(* CODESYS project cl_errorsdatabaseplc.library
   Company: CleanGreensSA
   Description: class to load error and class messages from SQL database
   Version: 1.0
   Placeholder: CL_errorDB
   Author: Martin Coffy and Massimo Lucano
   Title: ErrorDatabase_class

Project tree, tasks and I/O mapping:
  libraries: Tc2_Database, * (Beckhoff Automation GmbH); Tc2_DataExchange, * (Beckhoff Automation GmbH); Tc2_Standard, * (Beckhoff Automation GmbH); Tc2_System, * (Beckhoff Automation GmbH); Tc2_Utilities, * (Beckhoff Automation GmbH); Tc3_Database, * (Beckhoff Automation GmbH); Tc3_EventLogger, * (Beckhoff Automation GmbH); Tc3_Module, * (Beckhoff Automation GmbH)
  DUTs/
    Database/
      data type Main_STM
      data type ST_classAndErrorNum
      data type ST_ErrorDBConst
      data type ST_ParameterValues
      data type ST_SP_ClassReturn
      data type ST_SP_RecordReturn
      data type ST_valToAccess
      data type STM_LoadDB
  GVLs/
    global variables C
  POUs/
    Classes_database_connection/
      function block CL_CGSDictionnary [ST]: Init, Search
      function block CL_ErrorDB [ST]: GetClassMsg, GetErrorLongMsg, GetErrorRemedMsg, GetErrorShortMsg, GetNumerics, Init, nextPower2, numIterations, Run, SearchClassData, SearchErrorData, sMsgLang, stConstValues, WhichSeverity
      function block FB_SP_getClassNameAndIDs [ST]
      function block FB_SP_getErrorsMessages [ST]
*)

// DUTs/Database/Main_STM
{attribute 'qualified_only'}
{attribute 'strict'}
TYPE Main_STM :
(
  Init,
  Run,
  FillingArrays,
  SearchIndex,
  Idle,
  Error
);
END_TYPE

// DUTs/Database/ST_classAndErrorNum
TYPE ST_classAndErrorNum :
	STRUCT
		errorId					: STRING(3);
		classId					: STRING(3);
		telegramSending	: STRING(1);
		hmiErrorShow		: STRING(1);
		instanceNum			: BYTE;
	END_STRUCT
END_TYPE

// DUTs/Database/ST_ErrorDBConst
TYPE ST_ErrorDBConst :
	STRUCT
		udiErrNumRecord		  :	UDINT := 0;
		udiClassNumRecord		:	UDINT := 0;
		sLanguageForErrors	:	STRING(2)	:= 'en';
		udiUsedDB						:	UDINT := 0;
		tDBConnectTimeout		:	TIME	:=	TIME#15S;
		tAMSTimeout					:	TIME	:=	TIME#10S;
	END_STRUCT
END_TYPE

// DUTs/Database/ST_ParameterValues
TYPE ST_ParameterValues :
STRUCT
	lang: STRING(2);
END_STRUCT
END_TYPE

// DUTs/Database/ST_SP_ClassReturn
TYPE ST_SP_ClassReturn :
STRUCT
	tableId: UDINT;
	classId: STRING(3);
	className: STRING(255);
	instanceNum: BYTE;
	objDescriptMsg:	STRING(255);
END_STRUCT
END_TYPE

// DUTs/Database/ST_SP_RecordReturn
TYPE ST_SP_RecordReturn :
STRUCT
	tableId: UDINT;
	//classId: STRING(3);
	errorId: STRING(3);
	severity: BYTE;
	errorMsgShort: STRING(255);
	errorMsgLong: STRING(255);
	remediationMsg: STRING(255);
	telegramSending: STRING(1);
	hmiErrorShow: STRING(1);
END_STRUCT
END_TYPE

// DUTs/Database/ST_valToAccess
TYPE ST_valToAccess :
STRUCT
  	severity: BYTE;
	errorSummary:	STRING(255);
	errorMessage: STRING(255);
	remediationMessage: STRING(255);
	telegramSending: STRING(1);
	hmiErrorShow: STRING(1);
END_STRUCT
END_TYPE

// DUTs/Database/STM_LoadDB
{attribute 'qualified_only'}
{attribute 'strict'}
TYPE STM_LoadDB :
(
  
  GetAMSAdress,
	StoreErrorView,
	StoreClassView,
  GenErrorKeys,
	GenClassKeys,
	EndReadingDB
);
END_TYPE

// GVLs/C
// constant to be set in order to describe the greenhouse
// abbreviation GH stands everywhere for Greenhouse
{attribute 'qualified_only'}
VAR_GLOBAL CONSTANT 
  //Errors database constants
  nMaxRecordsDb_C          : UDINT := 1024;
  nMaxUpSize_C             : UDINT := 2048;
  //uiErrorUpSizePowerTwo_C : UDINT := 1024;
  //uiClassUpSizePowerTwo_C : UDINT := 1024;
END_VAR

// POUs/Classes_database_connection/CL_CGSDictionnary
FUNCTION_BLOCK CL_CGSDictionnary
VAR
	bInit	            :	BOOL	:= FALSE;
	
	_usiNbIter_C	    :	USINT;
	_udiSizeKeyArray	:	UDINT;
	
	usiSearchIter     : USINT;
  udiUpId           : UDINT;
  udiDownId         : UDINT;
	
	// Pointer to the keys array to search into
	_udiKeyArray_P	:	POINTER TO UDINT;	// Access to the keys array with a pointer, limited risks as long as udiUpId and udiDownId are correctly set.
END_VAR

METHOD PUBLIC Init : BOOL
VAR_INPUT
	udiKeyArray_P		:	POINTER TO UDINT;
	usiNbIter_C			:	SINT;
	udiSizeKeyArray	:	UDINT;
END_VAR

VAR
	bInputContract 	: BOOL;
END_VAR
Init := FALSE;

IF NOT bInit THEN
		
	bInputContract := 		udiKeyArray_P <> 0
										AND usiNbIter_C > 0 
										AND LREAL_TO_UDINT(EXPT(2,usiNbIter_C)) = udiSizeKeyArray;	// For the real size of the array, to do it outside (too complicated here)
	
	IF bInputContract THEN	// Test for the size of the inputs: to check if possible 
		
		// Initialisation of the "constant" values
		_udiKeyArray_P		:= udiKeyArray_P;
		_usiNbIter_C			:=	usiNbIter_C;
		_udiSizeKeyArray	:= udiSizeKeyArray;
		
		// Initialisation for the method
		usiSearchIter := usiNbIter_C;
  	udiUpId       := udiSizeKeyArray;
  	udiDownId     := 1;
		bInit := TRUE;
	END_IF
END_IF
END_METHOD

METHOD Search : BOOL
VAR_INPUT
  udiKey_DB	:	UDINT	:=	0;
END_VAR
VAR_OUTPUT
	udiFoundKeyIndex	:	UDINT;
  bError:  BOOL;
END_VAR
VAR
  udiMidDownId: UDINT;
  udiMidUpId: UDINT;
  udiMidUpKey: UDINT;
  udiMidLowKey:  UDINT;
END_VAR
IF bInit THEN

  Search := FALSE; 
  bError := FALSE;
  
  udiMidDownId := (udiUpId+udiDownId-1)/2;
  udiMidUpId := udiMidDownId+1;
      
  udiMidUpKey := _udiKeyArray_P[udiMidUpId];
  udiMidLowKey := _udiKeyArray_P[udiMidDownId];
      
  // Also manage the case when final iter and no case found
  IF udiKey_DB = udiMidLowKey THEN
		udiFoundKeyIndex := udiMidDownId+1;	// +1 required, since the Pointer index begins at 0, while the corresponding array starts at 1!
		usiSearchIter := _usiNbIter_C;
		udiUpId   := _udiSizeKeyArray;
		udiDownId := 1;
    Search := TRUE;
  ELSIF udiMidUpKey = udiKey_DB THEN
		udiFoundKeyIndex := udiMidUpId+1;	//+1 required, since the Pointer index begins at 0, while the corresponding array starts at 1!
		usiSearchIter := _usiNbIter_C;
		udiUpId   := _udiSizeKeyArray;
		udiDownId := 1;
    Search	:= TRUE;
  ELSE 
    IF usiSearchIter > 1 THEN
      IF udiMidLowKey > udiKey_DB THEN
          udiUpId := udiMidDownId;
					usiSearchIter := usiSearchIter-1;
      ELSIF udiMidUpKey < udiKey_DB THEN
          udiDownId := udiMidUpId;
					usiSearchIter := usiSearchIter-1;
      ELSE
				usiSearchIter := _usiNbIter_C;
				udiUpId   := _udiSizeKeyArray;
				udiDownId := 1;
				Search := TRUE;
				bError := TRUE;
      END_IF
    ELSE
			usiSearchIter := _usiNbIter_C;
			udiUpId   := _udiSizeKeyArray;
			udiDownId := 1;
      Search := TRUE;
      bError := TRUE;
    END_IF
  END_IF
END_IF
END_METHOD

END_FUNCTION_BLOCK

// POUs/Classes_database_connection/CL_ErrorDB
FUNCTION_BLOCK CL_ErrorDB
VAR  
  // Internal variables
  bInit                   :	BOOL	:= FALSE;
  stmMain                 : Main_STM := Main_STM.Init;
	
	// AMS variable
	fbAMSaddrGetter	        :	FB_GetLocalAmsNetId;
  
  // DB related variables
  // langStruct: ST_ParameterValues := (lang := C.sLangErrors);
  dbErrorConnector        : FB_SP_getErrorsMessages;
	dbClassConnector        :	FB_SP_getClassNameAndIDs;
  stmLoadDB               : STM_LoadDB	:= STM_LoadDB.GetAMSAdress;
  udiIndex                : UDINT := 1;
  
  // Size-related variables (previously known)
  _stError_ARP  	        : POINTER TO ARRAY [1..C.nMaxRecordsDb_C] OF ST_SP_RecordReturn;
  _sizeOfstError_AR       : UDINT;
	_stClass_ARP		        : POINTER TO ARRAY [1..C.nMaxRecordsDb_C] OF ST_SP_ClassReturn;
  _sizeOfstClass_AR       : UDINT;
	
  //udiErrorKeys_ARP        : ARRAY[1..C.nMaxUpSize_C] OF UDINT := [C.nMaxUpSize_C(0)];
	//udiClassKeys_ARP		    :	ARRAY[1..C.nMaxUpSize_C] OF UDINT := [C.nMaxUpSize_C(0)];

  udiErrorKeys_ARP        : POINTER TO ARRAY[1..C.nMaxUpSize_C] OF UDINT;
	udiClassKeys_ARP		    :	POINTER TO ARRAY[1..C.nMaxUpSize_C] OF UDINT;
	
	// Dictionnary objects - used to generalised the key search to any type of data structure
	objErrorDict	          :	CL_CGSDictionnary;
	objClassDict	          :	CL_CGSDictionnary;
	
	// Variables containing constants
  _uiClassShiftIndex      : UDINT;
  _uiErrShiftIndex        : UDINT;
  _uiUpSizeErrPowerTwo    : UDINT;
  _uiUpSizeClassPowerTwo  : UDINT;
  _uiErrNumIter           : SINT;
  _uiClassNumIter         : SINT;
	_stConstValues	        :	ST_ErrorDBConst;
	
	// AMS address
	sAMSAdrDbConnect        :	T_AmsNetId;
	stLangMsg               :	ST_ParameterValues	:= (lang := '');	//:= (lang := C.sLangErrors);
END_VAR

METHOD PUBLIC GetClassMsg : STRING(255)
VAR_INPUT
	udiIndex	:	UDINT;
END_VAR
GetClassMsg := _stClass_ARP^[udiIndex].objDescriptMsg;
END_METHOD

METHOD PUBLIC GetErrorLongMsg : STRING(255)
VAR_INPUT
	udiIndex	:	UDINT;
END_VAR
GetErrorLongMsg := _stError_ARP^[udiIndex].errorMsgLong;
END_METHOD

METHOD PUBLIC GetErrorRemedMsg : STRING(255)
VAR_INPUT
	udiIndex	:	UDINT;
END_VAR
GetErrorRemedMsg := _stError_ARP^[udiIndex].remediationMsg;
END_METHOD

METHOD PUBLIC GetErrorShortMsg : STRING(255)
VAR_INPUT
	udiIndex	:	UDINT;
END_VAR
GetErrorShortMsg := _stError_ARP^[udiIndex].errorMsgShort;
END_METHOD

METHOD PUBLIC GetNumerics : ST_classAndErrorNum
VAR_INPUT
	udiErrorIndex	:	UDINT;
	udiClassIndex	:	UDINT;
END_VAR
GetNumerics.errorId := _stError_ARP^[udiErrorIndex].errorId;
GetNumerics.hmiErrorShow	:=	_stError_ARP^[udiErrorIndex].hmiErrorShow;
GetNumerics.telegramSending := _stError_ARP^[udiErrorIndex].telegramSending;
GetNumerics.classId := _stClass_ARP^[udiClassIndex].classId;
GetNumerics.instanceNum := _stClass_ARP^[udiClassIndex].instanceNum;
END_METHOD

METHOD PUBLIC Init : BOOL
VAR_INPUT
  stConstValues   : ST_ErrorDBConst;
END_VAR
VAR
	structSize			: UINT;
	arraySize				: UDINT;
  ind             : UDINT;
END_VAR
_stConstValues := stConstValues;
Init := bInit := FALSE;
IF _stConstValues.udiUsedDB > 0 AND (_stConstValues.udiErrNumRecord > 0) AND (_stConstValues.udiErrNumRecord < C.nMaxRecordsDb_C) AND (_stConstValues.udiClassNumRecord > 0) AND (_stConstValues.udiClassNumRecord < C.nMaxRecordsDb_C) THEN
  _uiUpSizeErrPowerTwo:= nextPower2(_stConstValues.udiErrNumRecord);
  _uiUpSizeClassPowerTwo := nextPower2(_stConstValues.udiClassNumRecord);

  _uiErrShiftIndex := _uiUpSizeErrPowerTwo - _stConstValues.udiErrNumRecord;
  _uiClassShiftIndex := _uiUpSizeClassPowerTwo - _stConstValues.udiClassNumRecord;

  _uiErrNumIter := DINT_TO_SINT(numIterations(_stConstValues.udiErrNumRecord));
  _uiClassNumIter := DINT_TO_SINT(numIterations(_stConstValues.udiClassNumRecord));
  
  //Errors DB array allocated in memory from 1..udiErrNumRecord
  structSize := SIZEOF(ST_SP_RecordReturn);
	arraySize := structSize * (_stConstValues.udiErrNumRecord+2);
  _sizeOfstError_AR := structSize * (_stConstValues.udiErrNumRecord+1);
	_stError_ARP := __NEW(BYTE, arraySize);

  //Classes DB array allocated in memory from 1..udiClassNumRecord
  structSize := SIZEOF(ST_SP_ClassReturn);
	arraySize := structSize * (_stConstValues.udiClassNumRecord+2);
  _sizeOfstClass_AR := structSize * (_stConstValues.udiClassNumRecord+1);
	_stClass_ARP := __NEW(BYTE, arraySize);
 
  IF _uiUpSizeErrPowerTwo < C.nMaxUpSize_C AND _uiUpSizeClassPowerTwo < C.nMaxUpSize_C THEN 
    //Errors Keys array allocated in memory from 1.._uiUpSizeErrPowerTwo
    structSize := SIZEOF(UDINT);
    arraySize := structSize * (_uiUpSizeErrPowerTwo+2);
    udiErrorKeys_ARP := __NEW(BYTE, arraySize);
    FOR ind := 1 TO _uiUpSizeErrPowerTwo DO
      udiErrorKeys_ARP^[ind] := 0;
		END_FOR
  
    //Classes Keys array allocated in memory from 1.._uiUpSizeClassPowerTwo
    structSize := SIZEOF(UDINT);
    arraySize := structSize * (_uiUpSizeClassPowerTwo+2);
    udiClassKeys_ARP := __NEW(BYTE, arraySize);
    FOR ind := 1 TO _uiUpSizeClassPowerTwo DO
      udiClassKeys_ARP^[ind] := 0;
		END_FOR
    
    Init := bInit := TRUE;
  END_IF
END_IF
END_METHOD

METHOD PRIVATE nextPower2 : UDINT
VAR_INPUT
  n : UDINT;
END_VAR
VAR
  power : UDINT := 1;
END_VAR
IF (n <= 0) THEN
  nextPower2 := 1;
ELSIF (n AND (n - 1)) = 0 THEN 
  // If n is already a power of 2
  nextPower2 := n;
ELSE

  WHILE (power < n) DO
     //power := SHL(power,1); // Left shift to get the next power of 2}
     power := power * 2;
  END_WHILE
   
  nextPower2 := power;
END_IF
END_METHOD

METHOD PRIVATE numIterations : DINT
VAR_INPUT
  size : UDINT;
END_VAR
VAR
  log2Size : REAL;
END_VAR
// Calculate the logarithm base 2 of the size
IF size > 0 THEN
    log2Size := LN(size) / LN(2.0);
    numIterations := TRUNC(log2Size) + 1;
ELSE
    numIterations := 0; // Handle invalid input
END_IF
END_METHOD

METHOD PUBLIC Run : BOOL
VAR_OUTPUT
  bLoadErr:  BOOL;
END_VAR
VAR
  bStillExec: BOOL;
	bAnError: BOOL;
END_VAR
IF NOT bInit THEN
  RETURN;
END_IF
 
Run := FALSE;
bLoadErr := FALSE;

CASE stmLoadDB OF
  STM_LoadDB.GetAMSAdress:	// Useless here, as the previous address was already given
    fbAMSaddrGetter(bExecute := TRUE, tTimeOut := _stConstValues.tAMSTimeout,bBusy => bStillExec, bError => bAnError, AddrString	=> sAMSAdrDbConnect);
      IF NOT bStillExec THEN
        IF bANError THEN
          Run := TRUE;
          bLoadErr := TRUE;
       ELSE
          stLangMsg.lang := _stConstValues.sLanguageForErrors;
          stmLoadDB := STM_LoadDB.StoreErrorView;
        END_IF
      END_IF

  STM_LoadDB.StoreErrorView:
    dbErrorConnector(sAMSNetId := sAMSAdrDbConnect,nDBID := _stConstValues.udiUsedDB, nRecordStartIndex := 0, nLengthRecord := _stConstValues.udiErrNumRecord,tTimeoutIn := _stConstValues.tDBConnectTimeout, sizeRecord := _sizeOfstError_AR, bExecute := TRUE, bBusy => bStillExec, bError => bAnError, stRecord_P := _stError_ARP, stParameterValues := stLangMsg); // tTimeout := T#30S
      IF NOT bStillExec THEN
        IF bANError THEN
          Run := TRUE;
          bLoadErr := TRUE;
        ELSE
          stmLoadDB := STM_LoadDB.StoreClassView;
        END_IF
      END_IF
      
  STM_LoadDB.StoreClassView:
    dbClassConnector(sAMSNetId := sAMSAdrDbConnect, nDBID := _stConstValues.udiUsedDB, nRecordStartIndex := 0, nLengthRecord := _stConstValues.udiClassNumRecord,tTimeoutIn := _stConstValues.tDBConnectTimeout, sizeRecord := _sizeOfstClass_AR, bExecute := TRUE, bBusy => bStillExec, bError => bAnError, stRecord_P := _stClass_ARP);
      IF NOT bStillExec THEN
        IF bANError THEN
          Run := TRUE;
          bLoadErr := TRUE;
        ELSE
          stmLoadDB := STM_LoadDB.GenErrorKeys;
        END_IF
      END_IF
  
  STM_LoadDB.GenErrorKeys:
//      udiErrorKeys_AR[udiIndex+ C.uiErrorShiftIndex_C] := STRING_TO_UDINT(_stError_ARP[udiIndex].errorId);	// error ID unique for any type of error, no matter the class!
    udiErrorKeys_ARP^[udiIndex+ _uiErrShiftIndex] := STRING_TO_UDINT(_stError_ARP^[udiIndex].errorId);	// error ID unique for any type of error, no matter the class!
    
    udiIndex := udiIndex + 1;
//      IF udiIndex > C.uiNumErrorSources_C THEN
    IF udiIndex > _stConstValues.udiErrNumRecord THEN
      udiIndex := 1;
//				objErrorDict.Init(udiKeyArray_P	:=	ADR(udiErrorKeys_AR),usiNbIter_C := C.uiErrorNumIter_C,udiSizeKeyArray := C.uiErrorUpSizePowerTwo_C);
      objErrorDict.Init(udiKeyArray_P	:=	udiErrorKeys_ARP,usiNbIter_C := _uiErrNumIter, udiSizeKeyArray := _uiUpSizeErrPowerTwo);
      stmLoadDB := STM_LoadDB.GenClassKeys;
    END_IF
    
STM_LoadDB.GenClassKeys:
//      udiClassKeys_AR[udiIndex+ C.uiClassShiftIndex_C] := STRING_TO_UDINT(_stClass_ARP[udiIndex].classId);	// error ID unique for any type of error, no matter the class!
    udiClassKeys_ARP^[udiIndex+ _uiClassShiftIndex] := STRING_TO_UDINT(_stClass_ARP^[udiIndex].classId);
    
    udiIndex := udiIndex + 1;
//      IF udiIndex > C.uiNumClassWithErr_C THEN
    IF udiIndex > _stConstValues.udiClassNumRecord THEN
      udiIndex := 1;
//				objClassDict.Init(udiKeyArray_P	:=	ADR(udiClassKeys_AR),usiNbIter_C := C.uiClassNumIter_C,udiSizeKeyArray := C.uiClassUpSizePowerTwo_C);
      objClassDict.Init(udiKeyArray_P	:=	udiClassKeys_ARP,usiNbIter_C := _uiClassNumIter, udiSizeKeyArray := _uiUpSizeClassPowerTwo);
      stmLoadDB := STM_LoadDB.EndReadingDB;  
    END_IF

STM_LoadDB.EndReadingDB:
  Run := TRUE;
  bInit := TRUE;
  bLoadErr := FALSE;
  stmLoadDB := STM_LoadDB.StoreErrorView;
  
END_CASE
END_METHOD

METHOD SearchClassData : BOOL
VAR_INPUT
  classID	:	STRING(3);
END_VAR
VAR_OUTPUT
//	values:	ST_SP_ClassReturn;
	udiClassIndex:	UDINT;
  error:  BOOL;
END_VAR
VAR
	bExecEnd:		BOOL;
	foundKey	:	UDINT;
	uiSafeIter:	USINT := 0;
END_VAR
REPEAT
	bExecEnd := objClassDict.Search(udiKey_DB := STRING_TO_UDINT(classID),udiFoundKeyIndex => foundKey, bError => error);
	uiSafeIter := uiSafeIter + 1;
//	UNTIL (bExecEnd = TRUE) OR (uiSafeIter > C.uiClassNumIter_C)
	UNTIL (bExecEnd = TRUE) OR (uiSafeIter > _uiClassNumIter)
END_REPEAT

//values := _stClass_ARP[foundKey-C.uiClassShiftIndex_C];
udiClassIndex := foundKey -_uiClassShiftIndex;
END_METHOD

METHOD SearchErrorData : BOOL
VAR_INPUT
  errorID	:	STRING(3);
END_VAR
VAR_OUTPUT
//	values:	ST_SP_RecordReturn;
	udiErrorIndex	:	UDINT;
  error:  BOOL;
END_VAR
VAR
	bExecEnd:		BOOL;
	foundKey	:	UDINT;
	uiSafeIter:	USINT := 0;
END_VAR
REPEAT
	bExecEnd := objErrorDict.Search(udiKey_DB := STRING_TO_UDINT(errorID),udiFoundKeyIndex => foundKey, bError => error);
	uiSafeIter := uiSafeIter + 1;
//	UNTIL (bExecEnd = TRUE) OR (uiSafeIter > C.uiErrorNumIter_C)
	UNTIL (bExecEnd = TRUE) OR (uiSafeIter > _uiErrNumIter)
END_REPEAT

//values := _stError_ARP[foundKey-C.uiErrorShiftIndex_C];
udiErrorIndex := foundKey-_uiErrShiftIndex;
END_METHOD

PROPERTY PUBLIC sMsgLang : STRING(2)
GET
sMsgLang := _stConstValues.sLanguageForErrors;
END_GET
END_PROPERTY

PROPERTY PUBLIC stConstValues : ST_ErrorDBConst
GET
stConstValues	:= _stConstValues;
END_GET
SET
_stConstValues	:= stConstValues;
END_SET
END_PROPERTY

METHOD PUBLIC WhichSeverity : BYTE
VAR_INPUT
	udiIndex	: UDINT;
END_VAR
WhichSeverity := _stError_ARP^[udiIndex].severity;
END_METHOD

END_FUNCTION_BLOCK

// POUs/Classes_database_connection/FB_SP_getErrorsMessages
FUNCTION_BLOCK FB_SP_getErrorsMessages
VAR_INPUT
	sAMSNetId	:	T_AmsNetId;
	nDBID	:	UDINT	:= 1;
	nRecordStartIndex: UDINT;
  nLengthRecord:     UDINT;
	tTimeoutIn: TIME;
	bExecute: BOOL;
  stRecord_P: POINTER TO ST_SP_RecordReturn;  // Modified by hand!
  sizeRecord: UDINT;
END_VAR
VAR_OUTPUT
	bBusy: BOOL;
	bError: BOOL;
	ipResult: I_TcMessage;
END_VAR
VAR_IN_OUT
	stParameterValues: ST_ParameterValues;
END_VAR
VAR
	R_TRIG_Execute: R_TRIG;
	nState: INT := 0;
	nErrState: INT;
//	fbSQLDatabase         : FB_SQLDatabaseEvt(sNetID := sAMSNetId, tTimeout := tTimeoutIn);
//	fbSQLStoredProcedure  : FB_SQLStoredProcedureEvt(sNetID := sAMSNetId, tTimeout := tTimeoutIn);
//	fbSQLResult           : FB_SQLResultEvt(sNetID := sAMSNetId, tTimeout := tTimeoutIn);
	fbSQLDatabase         : FB_SQLDatabaseEvt(sNetID := '', tTimeout := T#15S);
	fbSQLStoredProcedure  : FB_SQLStoredProcedureEvt(sNetID := '', tTimeout := T#15S);
	fbSQLResult           : FB_SQLResultEvt(sNetID := '', tTimeout := T#15S);
	arrParaInfo           : ARRAY[0..0] OF ST_SQLSPParameter;
	
END_VAR

CASE nState OF
	0:
		R_TRIG_Execute(CLK:=bExecute);
		IF R_TRIG_Execute.Q THEN
			nState := 1;
			bBusy:=TRUE;
			bError:=FALSE;
			nErrState:=0;
		END_IF
	1:
		IF fbSQLDatabase.Connect(nDBID) THEN
			ipResult:=fbSQLDatabase.ipTcResult;
			IF fbSQLDatabase.bError THEN
				nErrState:=1;
				nState:=255;
			ELSE
				arrParaInfo[0].sParameterName := 'lang';
				arrParaInfo[0].eParameterType := E_SPParameterType.Input;
				arrParaInfo[0].eParameterDataType := E_ColumnType.NChar;
				arrParaInfo[0].nParameterSize := 3;

				nState:= 2;
			END_IF
		END_IF
	2:
		IF fbSQLDatabase.CreateSP('plcGetConfig', ADR(arrParaInfo), SIZEOF(arrParaInfo), ADR(fbSQLStoredProcedure)) THEN
			IF fbSQLDatabase.bError THEN
				nErrState:=2;
				nState:=255;
			ELSE
				nState:=3;
			END_IF
		END_IF
	3:
		IF fbSQLStoredProcedure.ExecuteDataReturn(ADR(stParameterValues), SIZEOF(stParameterValues), ADR(fbSQLResult))THEN
			ipResult:=fbSQLStoredProcedure.ipTcResult;
			IF fbSQLStoredProcedure.bError THEN
				nErrState:=3;
				nState:=255;
			ELSE
				nState:= 4;
			END_IF
		END_IF
	4:
		IF fbSQLResult.Read(nRecordStartIndex, nLengthRecord, stRecord_P, sizeRecord, FALSE, TRUE) THEN
			ipResult:=fbSQLResult.ipTcResult;
			IF fbSQLResult.bError THEN
				nErrState:=4;
				nState:= 255;
			ELSE
				nState:= 5;
			END_IF
		END_IF
	5:
		IF fbSQLStoredProcedure.Release() THEN
			IF fbSQLStoredProcedure.bError THEN
				nErrState:=5;
				nState:=255;
			ELSE
				nState:= 200;
			END_IF
		END_IF
	200:
		IF fbSQLDatabase.Disconnect() THEN
			nState := 0;
			bBusy:= FALSE;
		END_IF
	255:
		bError:= TRUE;
		bBusy:= FALSE;
		IF nErrState > 1 THEN
			nState:=200;
		ELSE
			nState:=0;
		END_IF
END_CASE

END_FUNCTION_BLOCK

// POUs/Classes_database_connection/FB_SP_getClassNameAndIDs
FUNCTION_BLOCK FB_SP_getClassNameAndIDs
VAR_INPUT
	sAMSNetId	:	T_AmsNetId;
	nDBID	:	UDINT	:= 1;
	nRecordStartIndex: UDINT;
	nLengthRecord:	UDINT;
	tTimeoutIn: TIME;
	bExecute: BOOL;
	stRecord_P: POINTER TO ST_SP_ClassReturn;
	sizeRecord: UDINT;
END_VAR
VAR_OUTPUT
	bBusy: BOOL;
	bError: BOOL;
	ipResult: I_TcMessage;
END_VAR
VAR
	R_TRIG_Execute: R_TRIG;
	nState: INT;
	nErrState: INT;
//	fbSQLDatabase: FB_SQLDatabaseEvt(sNetID := sAMSNetId, tTimeout := tTimeoutIn);
//	fbSQLStoredProcedure: FB_SQLStoredProcedureEvt(sNetID := sAMSNetId, tTimeout := tTimeoutIn);
//	fbSQLResult: FB_SQLResultEvt(sNetID := sAMSNetId, tTimeout := tTimeoutIn);
	fbSQLDatabase: FB_SQLDatabaseEvt(sNetID := '', tTimeout := T#15S);
	fbSQLStoredProcedure: FB_SQLStoredProcedureEvt(sNetID := '', tTimeout := T#15S);
	fbSQLResult: FB_SQLResultEvt(sNetID := '', tTimeout := T#15S);
END_VAR

CASE nState OF
	0:
		R_TRIG_Execute(CLK:=bExecute);
		IF R_TRIG_Execute.Q THEN
			nState := 1;
			bBusy:=TRUE;
			bError:=FALSE;
			nErrState:=0;
		END_IF
	1:
		IF fbSQLDatabase.Connect(hDBID := nDBID) THEN
			ipResult:=fbSQLDatabase.ipTcResult;
			IF fbSQLDatabase.bError THEN
				nErrState:=1;
				nState:=255;
			ELSE
				nState:= 2;
			END_IF
		END_IF
	2:
		IF fbSQLDatabase.CreateSP('getClassNameAndIDs', 0, 0, ADR(fbSQLStoredProcedure)) THEN
			IF fbSQLDatabase.bError THEN
				nErrState:=2;
				nState:=255;
			ELSE
				nState:=3;
			END_IF
		END_IF
	3:
		IF fbSQLStoredProcedure.ExecuteDataReturn(0, 0, ADR(fbSQLResult))THEN
			ipResult:=fbSQLStoredProcedure.ipTcResult;
			IF fbSQLStoredProcedure.bError THEN
				nErrState:=3;
				nState:=255;
			ELSE
				nState:= 4;
			END_IF
		END_IF
	4:
		IF fbSQLResult.Read(nRecordStartIndex, nLengthRecord,stRecord_P, sizeRecord, FALSE, TRUE) THEN
			ipResult:=fbSQLResult.ipTcResult;
			IF fbSQLResult.bError THEN
				nErrState:=4;
				nState:= 255;
			ELSE
				nState:= 5;
			END_IF
		END_IF
	5:
		IF fbSQLStoredProcedure.Release() THEN
			IF fbSQLStoredProcedure.bError THEN
				nErrState:=5;
				nState:=255;
			ELSE
				nState:= 200;
			END_IF
		END_IF
	200:
		IF fbSQLDatabase.Disconnect() THEN
			nState := 0;
			bBusy:= FALSE;
		END_IF
	255:
		bError:= TRUE;
		bBusy:= FALSE;
		IF nErrState > 1 THEN
			nState:=200;
		ELSE
			nState:=0;
		END_IF
END_CASE

END_FUNCTION_BLOCK
